VAR_GLOBAL CONSTANT
	nEndOfNodeIDVarsArray_2Dim: UINT := 9;
	nArrayTestLength_2DimX: UDINT := 4;
	nArrayTestLength_2DimY: UDINT := 2;
	//nArrayTestLength_2DimX*nArrayTestLength_2DimY*80
	nMaxReadDataArray_2Dim: UDINT := 640; 
	//sOpcUA_URL: STRING := 'opc.tcp://henningm-nb:4840';
	sOpcUA_URL: STRING := 'opc.tcp://localhost:4842';
	sNodeIDNamespace: STRING := 'TmcPLC';
END_VAR
VAR_GLOBAL
	NodeID_Identifiers: ARRAY[0..nEndOfNodeIDVarsArray_2Dim] OF STRING := 
		['GVL_ArrayTests2DimPLC.stat_BOOL_2Dim', 
		 'GVL_ArrayTests2DimPLC.stat_BSTRARRAY_2Dim',
		 'GVL_ArrayTests2DimPLC.stat_I1_2Dim', 
		 'GVL_ArrayTests2DimPLC.stat_I2_2Dim', 
		 'GVL_ArrayTests2DimPLC.stat_I4_2Dim', 
		 'GVL_ArrayTests2DimPLC.stat_R8_2Dim', 
		 'GVL_ArrayTests2DimPLC.stat_UI1_2Dim', 
		 'GVL_ArrayTests2DimPLC.stat_UI2_2Dim', 
		 'GVL_ArrayTests2DimPLC.stat_UI4_2Dim',
		 'GVL_ArrayTests2DimPLC.stat_DATE_2Dim'
	];
	NodeID_Sizes: ARRAY[0..nEndOfNodeIDVarsArray_2Dim] OF UDINT := 
		[(1 * nArrayTestLength_2DimX * nArrayTestLength_2DimY), 
		 (81 * nArrayTestLength_2DimX * nArrayTestLength_2DimY), 
		 (1 * nArrayTestLength_2DimX * nArrayTestLength_2DimY), 
		 (2 * nArrayTestLength_2DimX * nArrayTestLength_2DimY), 
		 (4 * nArrayTestLength_2DimX * nArrayTestLength_2DimY), 
		 (8 * nArrayTestLength_2DimX * nArrayTestLength_2DimY), 
		 (1 * nArrayTestLength_2DimX * nArrayTestLength_2DimY), 
		 (2 * nArrayTestLength_2DimX * nArrayTestLength_2DimY), 
		 (4 * nArrayTestLength_2DimX * nArrayTestLength_2DimY), 
		 (4 * nArrayTestLength_2DimX * nArrayTestLength_2DimY)
	];
	NodeID_DoOrDont: ARRAY[0..nEndOfNodeIDVarsArray_2Dim] OF BOOL := 
		[TRUE, //'GVL_ArrayTests3DimPLC.stat_BOOL_3Dim', 
		 TRUE, //'GVL_ArrayTests3DimPLC.stat_BSTRARRAY_3Dim',
		 TRUE, //'GVL_ArrayTests3DimPLC.stat_I1_3Dim', 
		 TRUE, //'GVL_ArrayTests3DimPLC.stat_I2_3Dim', 
		 TRUE, //'GVL_ArrayTests3DimPLC.stat_I4_3Dim', 
		 TRUE, //'GVL_ArrayTests3DimPLC.stat_R8_3Dim', 
		 TRUE, //'GVL_ArrayTests3DimPLC.stat_UI1_3Dim', 
		 TRUE, //'GVL_ArrayTests3DimPLC.stat_UI2_3Dim',  
		 TRUE, //'GVL_ArrayTests3DimPLC.stat_UI4_3Dim', 
		 FALSE //'GVL_ArrayTests3DimPLC.stat_DATE_3Dim'
	];
	NodeID_WriteCommands: ARRAY[0..nEndOfNodeIDVarsArray_2Dim] OF U_Arrays2DimInOne := [
			(bBool := [TRUE, FALSE, TRUE, FALSE, TRUE, FALSE, TRUE, FALSE]), 
	 		(sString := ['aaa', 'bbbb', 'ccccc', 'ddddddd', 'aaa', 'bbbb', 'ccccc', 'ddddddd']), 
			(bByte := [123, 124, 125, 126, 123, 124, 125, 126]), 
			(nInt := [127, 128, 129, 130,127, 128, 129, 130]), 
			(nUdint := [131, 132, 133, 134, 131, 132, 133, 134]), 
			(nLReal := [1.23456, 1.23457, 1.23458, 1.23459, 1.23456, 1.23457, 1.23458, 1.23459]), 
			(bByte := [111, 112, 113, 114, 111, 112, 113, 114]), 
			(nInt := [115, 116, 117, 118,115, 116, 117, 118]), 
			(nUdint := [119, 120, 121, 122, 119, 120, 121, 122]), 
			(dDate := [DT#2008-9-26-0:11:12, DT#2008-9-26-0:11:13, DT#2008-9-26-0:11:14, DT#2008-9-26-0:11:15, DT#2008-9-26-0:11:12, DT#2008-9-26-0:11:13, DT#2008-9-26-0:11:14, DT#2008-9-26-0:11:15]) 
	];
	NodeID_ReadResults: ARRAY[0..nEndOfNodeIDVarsArray_2Dim] OF U_Arrays2DimInOne;
	NodeID_ReadWrittenResults: ARRAY[0..nEndOfNodeIDVarsArray_2Dim] OF U_Arrays2DimInOne;
	NodeID_CheckReadWrite: ARRAY[0..nEndOfNodeIDVarsArray_2Dim] OF BOOL;
	
	//Data fields
	stat_BOOL_2Dim: 		ARRAY[1..nArrayTestLength_2DimX, 1..nArrayTestLength_2DimY] OF BOOL 	:= [TRUE, TRUE, TRUE, TRUE, FALSE, FALSE, FALSE, FALSE]; 						(*~ (OPC : 1 : enabled for OPC) *)
	stat_BSTRARRAY_2Dim: 	ARRAY[1..nArrayTestLength_2DimX, 1..nArrayTestLength_2DimY] OF STRING 	:= ['these', 'are', 'init', 'values', 'which', 'will', 'be', 'overwritten'];	(*~ (OPC : 1 : enabled for OPC) *)
	stat_I1_2Dim: 			ARRAY[1..nArrayTestLength_2DimX, 1..nArrayTestLength_2DimY] OF BYTE		:= [1, 1, 1, 1, 1, 1, 1, 1];													(*~ (OPC : 1 : enabled for OPC) *)
	stat_I2_2Dim: 			ARRAY[1..nArrayTestLength_2DimX, 1..nArrayTestLength_2DimY] OF INT		:= [1, 1, 1, 1, 1, 1, 1, 1];													(*~ (OPC : 1 : enabled for OPC) *)
	stat_I4_2Dim:			ARRAY[1..nArrayTestLength_2DimX, 1..nArrayTestLength_2DimY] OF DINT 	:= [1, 1, 1, 1, 1, 1, 1, 1];													(*~ (OPC : 1 : enabled for OPC) *)
	stat_R8_2Dim: 			ARRAY[1..nArrayTestLength_2DimX, 1..nArrayTestLength_2DimY] OF LREAL	:= [1.1, 1.1, 1.1, 1.1, 1.1, 1.1, 1.1, 1.1];									(*~ (OPC : 1 : enabled for OPC) *)
	stat_UI1_2Dim:			ARRAY[1..nArrayTestLength_2DimX, 1..nArrayTestLength_2DimY] OF BYTE		:= [1, 1, 1, 1, 1, 1, 1, 1];													(*~ (OPC : 1 : enabled for OPC) *)
	stat_UI2_2Dim: 			ARRAY[1..nArrayTestLength_2DimX, 1..nArrayTestLength_2DimY] OF UINT		:= [1, 1, 1, 1, 1, 1, 1, 1];													(*~ (OPC : 1 : enabled for OPC) *)
	stat_UI4_2Dim: 			ARRAY[1..nArrayTestLength_2DimX, 1..nArrayTestLength_2DimY] OF UDINT	:= [1, 1, 1, 1, 1, 1, 1, 1];													(*~ (OPC : 1 : enabled for OPC) *)
	stat_DATE_2Dim:			ARRAY[1..nArrayTestLength_2DimX, 1..nArrayTestLength_2DimY] OF DT		:= [DT#2014-2-20-0:11:12, DT#2014-2-20-0:11:12, DT#2014-2-20-0:11:12, DT#2014-2-20-0:11:12, DT#2014-2-20-0:11:12, DT#2014-2-20-0:11:12, DT#2014-2-20-0:11:12, DT#2014-2-20-0:11:12];													(*~ (OPC : 1 : enabled for OPC) *)
		
END_VAR

(* stored: Version 1.1.0.1, ProductVersion 3.1.0.24
   GVL GVL_ArrayTests2DimPLC: Id {c803cc16-c8fe-45ce-ae95-618db4261664} *)
